Omron CX-Programmer project NewProject (CX-Programmer 9.51)

# PLC NewPLC1: CP1L L
; My_First_Project

## Program NewProgram1 (cyclic task 0)
Local symbols
button_1 0.00 BOOL
out_1 100.00 BOOL

### Section Section1

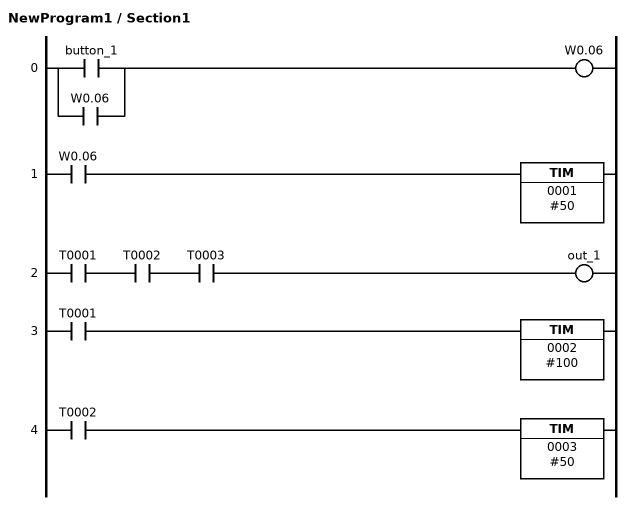
; rung 0
LD button_1
OR W0.06
OUT W0.06
; rung 1
LD W0.06
TIM 0001 #50
; rung 2
LD T0001
AND T0002
AND T0003
OUT out_1
; rung 3
LD T0001
TIM 0002 #100
; rung 4
LD T0002
TIM 0003 #50

### Section END
; rung 0
END(001)